# B&R Automation Studio project PrintMarkLabWork
Automation Studio 4.12.4.107 SP; technology packages: Acp10Arnc0 5.23.1, mapp 5.23.1, mappView 5.23.0

## Configuration Config1

CPU X20CP0484, AutomationRuntime G4.93, Build 4.1.2, Vc V4.73.0

### Task classes (Cpu.sw)
```
Cyclic#1 (cycle 2000 us, tolerance 10000 us):
  AutoCtrl <- Source.AutoCtrl.AutoCtrl.prg  // Auto Ctrl Logic
  ConvCtrl <- Source.AxisConf.ConvCtrl.prg  // Conv Ctrl Logic
  CutterCtrl <- Source.AxisConf.CutterCtrl.prg  // Cutter Ctrl Logic
Cyclic#4 (cycle 100000 us, tolerance 100000 us):
  Alarm <- InfraStructure.Alarm.Alarm.prg  // Alarm Logic
Cyclic#7 (cycle 1000000 us, tolerance 1000000 us):
  Visu <- InfraStructure.Visu.Visu.prg  // Visu Logic
DataObjects: Acp10sys
NcDataObjects: acp10etxen <- Axis.acp10etxen.dob, gAxis01a <- Axis.gAxis01obj.gAxis01a.dob, gAxis01i <- Axis.gAxis01obj.gAxis01i.dob, gAxis02a <- Axis.gAxis02obj.gAxis02a.dob, gAxis02i <- Axis.gAxis02obj.gAxis02i.dob
Binaries: arsvcreg, udbdef, mvLoader, FWRules, TCData, TCLang, arflatprv, arcoal, Acp10map, acp10cfg, SlaveAxis, ashwac, User, sysconf, asfw, arconfig, ashwd, MasterAxis, iomap, Role, DataRConf, AlarmConf, UserConf, User_1, TC
Libraries: Acp10man, Acp10par, NcGlobal, Acp10_MC, sys_lib, brsystem, runtime, MpAxis, MpBase, MpCom, MpServer, MC_RegMa, MpAlarmX, astime, MpData, FileIO, DataObj, MpUserX, arssl, asieccon, powerlnk, asbrstr, aruser, arcert, aseth, ashw
```

### Hardware
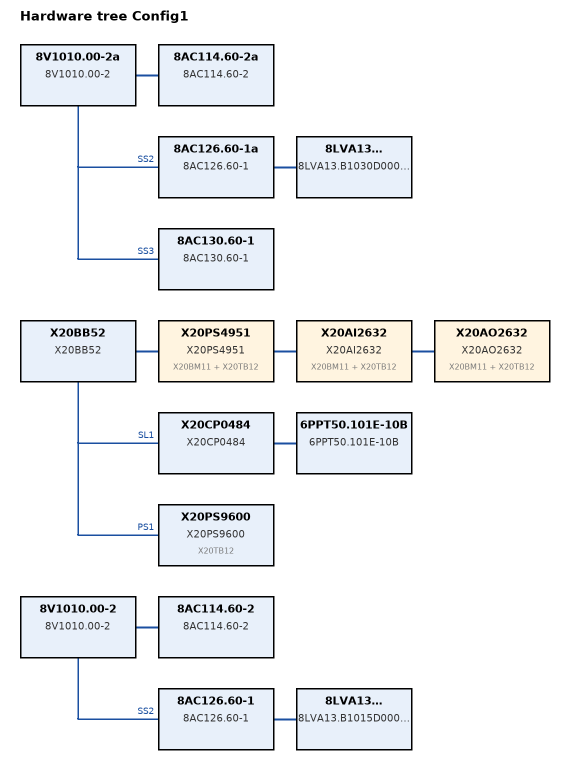
```
6PPT50.101E-10B : 6PPT50.101E-10B v1.3.8.0  [ETH1 -> X20CP0484.IF2 [Cable Type=PowerlinkCable, Length=10, Version=1.0.0.3]]
  Terminal = true
  Startmode = 2
  ShowBootlogoWeb = 1
  TimeZone = 250
  PasswordVNC = 
  BrowserVKeyboard = 0
  PasswordCIFS = 
  PasswordService = 
8AC114.60-2 : 8AC114.60-2 v1.0.0.8  [SS -> 8V1010.00-2.SS1; PLK1 -> X20CP0484.IF3 (NodeNumber=1) [Cable Type=PowerlinkCable, Length=10, Version=1.0.0.3]; PLK2 -> 8AC114.60-2a.PLK1 (NodeNumber=1) [Cable Type=PowerlinkCable, Length=10, Version=1.0.0.3]]
8AC114.60-2a : 8AC114.60-2 v1.0.0.8  [SS -> 8V1010.00-2a.SS1; PLK1 -> 8AC114.60-2.PLK2 (NodeNumber=2) [Cable Type=PowerlinkCable, Length=10, Version=1.0.0.3]]
8AC126.60-1 : 8AC126.60-1 v2.2.0.0  [SS -> 8V1010.00-2.SS2]
8AC126.60-1a : 8AC126.60-1 v2.2.0.0  [SS -> 8V1010.00-2a.SS2]
8AC130.60-1 : 8AC130.60-1 v2.2.0.0  [SS -> 8V1010.00-2a.SS3]
8LVA13.B1015D000-0 : 8LVA13.B1015D000-0 v2.2.0.3  [EC -> 8AC126.60-1.EC; MT -> 8V1010.00-2.MT1]
8LVA13.B1030D000-0 : 8LVA13.B1030D000-0 v2.2.0.3  [EC -> 8AC126.60-1a.EC; MT -> 8V1010.00-2a.MT1]
8V1010.00-2 : 8V1010.00-2 v2.2.0.0
  MotionTP = Acp10Arnc0
  SinglePhaseOperation = on
  BothEndSwitchesAreNormallyOpen_r1 = on
  QuickStopIsNormallyOpen_r1 = on
8V1010.00-2a : 8V1010.00-2 v2.2.0.0
  MotionTP = Acp10Arnc0
  SinglePhaseOperation = on
  AxisIsPeriodic_r1 = on
  Period_r1 = 3600
  BothEndSwitchesAreNormallyOpen_r1 = on
  QuickStopIsNormallyOpen_r1 = on
X20AI2632 : X20AI2632 v1.3.0.0  [SS1 -> X20TB12b.SS; SL -> X20BM11a.SL1]
  Supervision = off
X20AO2632 : X20AO2632 v1.2.0.0  [SS1 -> X20TB12c.SS; SL -> X20BM11b.SL1]
  Supervision = off
X20BB52 : X20BB52 v1.2.0.0
X20BM11 : X20BM11 v1.1.0.0  [X2X1 -> X20BB52.IF6]
X20BM11a : X20BM11 v1.1.0.0  [X2X1 -> X20BM11.X2X2]
X20BM11b : X20BM11 v1.1.0.0  [X2X1 -> X20BM11a.X2X2]
X20CP0484 : X20CP0484 v1.6.0.0  [SL -> X20BB52.SL1]
  Connector IF2:
    ActivateDevice = 1
    Mode = Manual
    InternetAddress = 10.91.10.142
    SubnetMask = 255.255.255.0
    ActivateSnmp = 2
  ConfigurationID = PrintMarkLabWork_Config1
  Simulation = 1
  TimerDeviceType = EPLX2X
  TimerDevice = X20CP0484.IF3
  TaskClassIdleTime = 2000
  Cyclic1Duration = 2000
  Cyclic1Tolerance = 10000
  Cyclic2Duration = 20000
  Cyclic2Tolerance = 20000
  Cyclic3Duration = 50000
  Cyclic3Tolerance = 50000
  Cyclic4Duration = 100000
  Cyclic4Tolerance = 100000
  Cyclic5Duration = 200000
  Cyclic5Tolerance = 200000
  Cyclic6Duration = 500000
  Cyclic6Tolerance = 500000
  Cyclic7Duration = 1000000
  Cyclic7Tolerance = 1000000
  Cyclic8Duration = 10000
  Cyclic8Tolerance = 30000000
  FileDevice1
  FileDeviceName1 = USER
  FileDevicePath1 = USER_PATH
  ActivateOpcUa = 1
  OpcUaInformationModels_PV_Version = 1
X20PS4951 : X20PS4951 v1.2.0.0  [SS1 -> X20TB12a.SS; SL -> X20BM11.SL1]
  Supervision = off
X20PS9600 : X20PS9600 v1.6.0.0  [PS -> X20BB52.PS1; SS1 -> X20TB12.SS]
X20TB12 : X20TB12 v1.0.0.0
X20TB12a : X20TB12 v1.0.0.0
X20TB12b : X20TB12 v1.0.0.0
X20TB12c : X20TB12 v1.0.0.0
```

### Acp10cfg.ncc - X20CP0484/Motion/Acp10cfg.ncc
```
NcConfiguration (Version=5.23.1, NcSwId=Acp10)
  ACP10CF1_typ:
    cnt_nettrc_rec_drive = 1500
    bufsize_trace_upload = 1200
    tc_nc_man_task = Cyclic #1
    glob_pv_as_ncobject = Yes
    ncsys_dl_broadcast = Yes
    ncsys_dl_acp_reset = Yes
    safemc_log_err_to_ax = Yes
    network_init:
      ncsw_init_execute = Yes
      automatic_execute = No
      node_nr_warning = Yes
      net_err_before_ncact = Yes
    nettrc:
      enter_parsecrec = Yes
      enter_ncaction = Yes
      save_ring_startidx = Yes
    cam_prof_download:
      cam_dat_dl_parallel = No
      tc_cam_dl_parallel = Task class for NC Manager task
    plk_if[0]:
      if_name = IF3
      tc_CycDat_PLCopen = Task class for NC Manager task
      mc_broadcast_extdat = No
```

### Acp10map.ncm - X20CP0484/Motion/Acp10map.ncm
```
NcMapping (NcSwId=Acp10, DisabledNodesAreHidden=False)
  NcObject gAxis01 (ModuleId=8V1010.00-2, Type=ncAXIS, Channel=1, AcoposSimulation=Off, InitParameter=gAxis01i, AcoposParameter=gAxis01a, Disabled=FALSE, ModuleDisabled=FALSE)
  NcObject 8V1010.00-2_ncV_AXIS1 (ModuleId=8V1010.00-2, Type=ncV_AXIS, Channel=1, Disabled=TRUE, ModuleDisabled=FALSE)
  NcObject gAxis02 (ModuleId=8V1010.00-2a, Type=ncAXIS, Channel=1, AcoposSimulation=Off, InitParameter=gAxis02i, AcoposParameter=gAxis02a, AdditionalData=PLCopen_ModPos="3600,1" , Disabled=FALSE, ModuleDisabled=FALSE)
  NcObject 8V1010.00-2a_ncV_AXIS1 (ModuleId=8V1010.00-2a, Type=ncV_AXIS, Channel=1, Disabled=TRUE, ModuleDisabled=FALSE)
```

### MasterAxis.mpaxisbasic - X20CP0484/Motion/MasterAxis.mpaxisbasic
```
Element gAxisMaster (Type=mpaxisbasic)
  Alarms = MpAlarmX
```

### SlaveAxis.mpaxisbasic - X20CP0484/Motion/SlaveAxis.mpaxisbasic
```
Element gAxisSlave (Type=mpaxisbasic)
  Alarms = MpAlarmX
```

### AlarmConf.mpalarmxcore - X20CP0484/mappServices/Alarm/AlarmConf.mpalarmxcore
```
Element gAlarmXMain (Type=mpalarmxcore)
  mapp.AlarmX.Core.Configuration:
    [0]:
      Name = InCuttingZone
      Message = Cutter is in Cutting Zone. Please Remove the Cutter
      Code = 50
      Severity = 10
      Behavior = PersistentAlarm
        ReactionUntilAcknowledged = FALSE
    [1]:
      Name = CuttingError
      Message = Product without Print Mark Exceeded Limit
      Code = 80
      Severity = 50
      Behavior = PersistentAlarm
        ReactionUntilAcknowledged = FALSE
```

### DataRConf.mpdatarecorder - X20CP0484/mappServices/DataRecorder/DataRConf.mpdatarecorder
```
Element gDataRecorder (Type=mpdatarecorder)
  Alarms = MpAlarmX
```

### UserConf.mpuserx - X20CP0484/mappServices/User/UserConf.mpuserx
```
Element UserMgmtX (Type=mpuserx)
  ServerSettings:
    Server:
      AdditionalUserData:
        [0] = mail
        [1] = telephoneNumber
  Users:
    DefUser#1:
      id = Admin
      name = Administrator
      lang = en
    DefUser#2:
      id = Operator
      name = Machine Operator
      lang = en
    DefUser#3:
      id = Anonymous
  Groups:
    DefGroup#1:
      id = Administrators
      level = 100
      admin = TRUE
      rights:
        [0] = FullAccess
    DefGroup#2:
      id = Operator
      level = 50
```

## Logical view

Binary libraries used (declarations not repeated): operator, runtime, astime, AsIecCon, Acp10man 5.23.1, Acp10par 5.23.1, NcGlobal 5.23.1, Acp10_MC 5.23.1, sys_lib, brsystem, MpAxis 1.86.0, MpBase, MpCom 5.23.1, MpServer, MC_RegMa 5.23.1, MpAlarmX 5.23.1, MpData 5.23.1, FileIO, DataObj, MpUserX 5.23.1

### Global.var - Global variables
```iecst
(*********************************************************************************
 * Copyright: B&R Industrial Automation GmbH
 * Author:    kasliwals
 * Created:   December 17, 2023/12:04 AM
 *********************************************************************************)
(*Axis Variables*)
VAR
	gAxis01 : ACP10AXIS_typ; (*Master Axis*)
	gAxis02 : ACP10AXIS_typ; (*Slave Axis*)
END_VAR
(*Axis Global structure*)
VAR
	gAx_Slave : AxisBasic_type; (*Slave Axis Structure*)
	gAx_Master : AxisBasic_type; (*MAster axis Structure*)
END_VAR
(*HMI Variables*)
VAR
	gMI_ModeConfirm : BOOL; (*Mode Confirm VA*)
	gMI_MODE : BOOL; (*Mode VA*)
END_VAR
```


### Package Logical/Axis - Axis Package

### Package Logical/Axis/gAxis01obj - gAxis01obj

### gAxis01i.ax
```
InitParameter (Version=5.23.1, NcSwId=ACP10)
  ACP10AXIS_typ:
    dig_in:
      level:
        reference = ncACTIV_HI
        pos_hw_end = ncACTIV_HI
        neg_hw_end = ncACTIV_HI
        trigger1 = ncACTIV_HI
        trigger2 = ncACTIV_HI
    encoder_if:
      parameter:
        count_dir = ncSTANDARD
        scaling:
          load:
            units = 1600
            rev_motor = 1
    limit:
      parameter:
        v_pos = 10000.0
        v_neg = 10000.0
        a1_pos = 50000.0
        a2_pos = 50000.0
        a1_neg = 50000.0
        a2_neg = 50000.0
        t_jolt = 0.0
        t_in_pos = 0.0
        pos_sw_end = 8388607
        neg_sw_end = -8388608
        ds_warning = 500.0
        ds_stop = 1000.0
        a_stop = 1.0E+30
        dv_stop = 0.0
        dv_stop_mode = ncOFF
    controller:
      mode = ncPOSITION + ncFF
      position:
        kv = 262.0
        tn = 0.0
        t_predict = 0.0004
        t_total = 0.0004
        p_max = 1.0E+30
        i_max = 0.0
      speed:
        kv = 0.55
        tn = 0.0
        t_filter = 0.0
        isq_filter1:
          type = ncOFF
          a0 = 0.0
          a1 = 0.0
          b0 = 0.0
          b1 = 0.0
          b2 = 0.0
          c0_par_id = 0
          c1_par_id = 0
        isq_filter2:
          type = ncOFF
          a0 = 0.0
          a1 = 0.0
          b0 = 0.0
          b1 = 0.0
          b2 = 0.0
          c0_par_id = 0
          c1_par_id = 0
        isq_filter3:
          type = ncOFF
          a0 = 0.0
          a1 = 0.0
          b0 = 0.0
          b1 = 0.0
          b2 = 0.0
          c0_par_id = 0
          c1_par_id = 0
      uf:
        type = ncLINEAR + ncCORRECTION
        auto_config = ncMOTOR_PAR
        u0 = 0.0
        un = 0.0
        fn = 50.0
        k_f_slip = 0.0
      ff:
        mode = ncSTANDARD
        torque_load = 0.0
        torque_pos = 0.0
        torque_neg = 0.0
        kv_torque = 0.0117175
        inertia = 8.74906E-05
        t_filter_a = 0.0
      fb:
        mode = ncSTANDARD
        speed_mix_ratio = 0.0
        speed_kv = 0.0
      model:
        mass1:
          inertia = 0.0
          viscous_friction = 0.0
        mass2:
          inertia = 0.0
          viscous_friction = 0.0
          stiffness = 0.0
          damping = 0.0
    move:
      stop:
        parameter[0]:
          decel_ramp = ncA_LIMIT
          controller = ncON
        parameter[1]:
          decel_ramp = ncA_LIMIT
          controller = ncON
        parameter[2]:
          decel_ramp = ncA_LIMIT
          controller = ncON
        parameter[3]:
          decel_ramp = ncA_LIMIT
          controller = ncON
        quickstop:
          decel_ramp = ncA_LIMIT
          t_jolt = 0.0
        drive_error:
          decel_ramp = ncA_LIMIT
      homing:
        parameter:
          s = 0
          v_switch = 5000.0
          v_trigger = 500.0
          a = 50000.0
          mode = ncDIRECT
          edge_sw = ncPOSITIVE
          start_dir = ncPOSITIVE
          trigg_dir = ncPOSITIVE
          ref_pulse = ncOFF
          fix_dir = ncOFF
          tr_s_block = 0.0
          torque_lim = 0.0
          ds_block = 0.0
          ds_stop = 0.0
      basis:
        parameter:
          v_pos = 500.0
          v_neg = 5000.0
          a1_pos = 50000.0
          a2_pos = 50000.0
          a1_neg = 50000.0
          a2_neg = 50000.0
    message:
      text:
        parameter:
          format = ncBREAK + ncZERO
          columns = 80
          data_modul = acp10etxen
```

### Package Logical/Axis/gAxis02obj - gAxis02obj

### gAxis02i.ax
```
InitParameter (Version=5.23.1, NcSwId=ACP10)
  ACP10AXIS_typ:
    dig_in:
      level:
        reference = ncACTIV_HI
        pos_hw_end = ncACTIV_HI
        neg_hw_end = ncACTIV_HI
        trigger1 = ncACTIV_HI
        trigger2 = ncACTIV_HI
    encoder_if:
      parameter:
        count_dir = ncSTANDARD
        scaling:
          load:
            units = 3600
            rev_motor = 1
    limit:
      parameter:
        v_pos = 108000.0
        v_neg = 108000.0
        a1_pos = 1080000.0
        a2_pos = 1080000.0
        a1_neg = 1080000.0
        a2_neg = 1080000.0
        t_jolt = 0.18
        t_in_pos = 0.0
        pos_sw_end = 8388607
        neg_sw_end = -8388608
        ds_warning = 180.0
        ds_stop = 360.0
        a_stop = 1.0E+30
        dv_stop = 0.0
        dv_stop_mode = ncOFF
    controller:
      mode = ncPOSITION + ncFF
      position:
        kv = 241.0
        tn = 0.0
        t_predict = 0.0004
        t_total = 0.0004
        p_max = 1.0E+30
        i_max = 0.0
      speed:
        kv = 0.55
        tn = 0.0
        t_filter = 0.0
        isq_filter1:
          type = ncOFF
          a0 = 0.0
          a1 = 0.0
          b0 = 0.0
          b1 = 0.0
          b2 = 0.0
          c0_par_id = 0
          c1_par_id = 0
        isq_filter2:
          type = ncOFF
          a0 = 0.0
          a1 = 0.0
          b0 = 0.0
          b1 = 0.0
          b2 = 0.0
          c0_par_id = 0
          c1_par_id = 0
        isq_filter3:
          type = ncOFF
          a0 = 0.0
          a1 = 0.0
          b0 = 0.0
          b1 = 0.0
          b2 = 0.0
          c0_par_id = 0
          c1_par_id = 0
      uf:
        type = ncLINEAR + ncCORRECTION
        auto_config = ncMOTOR_PAR
        u0 = 0.0
        un = 0.0
        fn = 50.0
        k_f_slip = 0.0
      ff:
        mode = ncSTANDARD
        torque_load = 0.0
        torque_pos = 0.0
        torque_neg = 0.0
        kv_torque = 0.00398844
        inertia = 0.00010255
        t_filter_a = 0.0
      fb:
        mode = ncSTANDARD
        speed_mix_ratio = 0.0
        speed_kv = 0.0
      model:
        mass1:
          inertia = 0.0
          viscous_friction = 0.0
        mass2:
          inertia = 0.0
          viscous_friction = 0.0
          stiffness = 0.0
          damping = 0.0
    move:
      stop:
        parameter[0]:
          decel_ramp = ncA_LIMIT
          controller = ncON
        parameter[1]:
          decel_ramp = ncA_LIMIT
          controller = ncON
        parameter[2]:
          decel_ramp = ncA_LIMIT
          controller = ncON
        parameter[3]:
          decel_ramp = ncA_LIMIT
          controller = ncON
        quickstop:
          decel_ramp = ncA_LIMIT
          t_jolt = 0.0
        drive_error:
          decel_ramp = ncA_LIMIT
      homing:
        parameter:
          s = 0
          v_switch = 5000.0
          v_trigger = 500.0
          a = 50000.0
          mode = ncDIRECT
          edge_sw = ncPOSITIVE
          start_dir = ncPOSITIVE
          trigg_dir = ncPOSITIVE
          ref_pulse = ncOFF
          fix_dir = ncOFF
          tr_s_block = 0.0
          torque_lim = 0.0
          ds_block = 0.0
          ds_stop = 0.0
      basis:
        parameter:
          v_pos = 500.0
          v_neg = 5000.0
          a1_pos = 50000.0
          a2_pos = 50000.0
          a1_neg = 50000.0
          a2_neg = 50000.0
    message:
      text:
        parameter:
          format = ncBREAK + ncZERO
          columns = 80
          data_modul = acp10etxen
```

### Package Logical/Source - Source Package

### Package Logical/Source/AutoCtrl - Auto Ctrl Package

### Program Logical/Source/AutoCtrl/AutoCtrl (IEC) - Auto Ctrl task

#### Main.st - Init, cyclic, exit code
```iecst
(*********************************************************************************
 * Copyright: B&R Industrial Automation GmbH
 * Author:    kasliwals
 * Created:   December 16, 2023/11:35 PM
* Description: Auto Ctrl Logic for Print Marl
* Version : 1.0.0.0
 *********************************************************************************)

PROGRAM _INIT
	(* Insert code here *)
	Status_CutterCtrl := PV_xgetadr(ADR('CutterCtrl:iCutterCtrl'),ADR(CutterAdd),ADR(SizeCutter));
	Status_ConvCtrl := PV_xgetadr(ADR('ConvCtrl:iConvCtrl'),ADR(ConvAdd),ADR(SizeConv));
	Status_CamSeq := PV_xgetadr(ADR('CutterCtrl:iAx_CamSeq'),ADR(CamAdd),ADR(SizeCam));
	Status_RegCapture := PV_xgetadr(ADR('CutterCtrl:iFb_RegCapture'),ADR(RegAdd),ADR(RegSize));
	gAx_Master.In.Enable := TRUE;
	gAx_Slave.In.Enable := TRUE;
	iMI_CurrentMode := 'Manual Mode';
END_PROGRAM

PROGRAM _CYCLIC
	(* Insert code here *)
	pCutterCtrl ACCESS CutterAdd;
	pConvCtrl ACCESS ConvAdd;
 	pAx_CamSeq ACCESS CamAdd;
	pRegCapture ACCESS RegAdd;

	CASE AutoCtrlState OF
		WAIT :
			iMI_MachineStatus := 'Please Select the Mode And Then Press Start';
			gAx_Master.In.Enable := TRUE;
			gAx_Slave.In.Enable := TRUE;

			IF iAutoCtrl.Cmd.Start THEN
				pConvCtrl.Cmd.Start := TRUE;
				pCutterCtrl.Cmd.Start := TRUE;
				AutoCtrlState := MODE_SELECT;
			END_IF

		MODE_SELECT :
			IF gMI_ModeConfirm THEN

				IF iAutoCtrl.Cmd.AutoMode THEN
					iMI_CurrentMode := 'Auto Mode';
					AutoCtrlState := HOMING_DONE;
				ELSE
					iMI_CurrentMode := 'Manual Mode';
					AutoCtrlState := MANUAL_START;
				END_IF
			END_IF
		HOMING_DONE :
			iMI_MachineStatus := 'Homing Both Axis';
			pAx_CamSeq.In.ErrorReset := TRUE;

			IF gAx_Master.Out.IsHomed AND gAx_Slave.Out.IsHomed THEN
				pAx_CamSeq.In.ErrorReset := FALSE;
				AutoCtrlState := AUTO_START;
			END_IF

		AUTO_START :

			IF pAx_CamSeq.Out.Info.MasterReady AND pAx_CamSeq.Out.Info.SlaveReady AND pAx_CamSeq.Out.StatusID = 0 THEN

				pAx_CamSeq.In.StartSequence := TRUE;
			END_IF
			IF pAx_CamSeq.Out.StatusID <> 0 THEN
				pAx_CamSeq.In.ErrorReset := TRUE;
				pAx_CamSeq.In.ErrorReset := FALSE;
			END_IF

			IF pAx_CamSeq.Out.InSync AND iAutoCtrl.Cmd.Start THEN
				iMI_MachineStatus := 'Running in Auto Mode';
				gAx_Master.In.MoveVelocity := TRUE;
			END_IF

			IF iAutoCtrl.Cmd.Stop THEN
				iMI_MachineStatus := 'Stop Pressed. Press Start to Restart Or Change mode to Exit Mode and select mode.';
				gAx_Master.In.MoveVelocity := FALSE;
			END_IF

			IF iAutoCtrl.Cmd.DisableCutter THEN
				iMI_MachineStatus := 'Cutter Disabled Pressed';
				pAx_CamSeq.In.StartSequence := FALSE;
				pCutterCtrl.Cmd.Start := FALSE;
				gAx_Slave.In.Power := FALSE;
				AutoCtrlState := CUTTER_DISABLED_HOME;
			END_IF

			IF iAutoCtrl.Cmd.ChangeMode AND iAutoCtrl.Cmd.Stop THEN
				iMI_MachineStatus := 'Machine Stopped';
				gAx_Master.In.MoveVelocity := FALSE;
				iAutoCtrl.Cmd.ChangeMode := FALSE;
				pAx_CamSeq.In.StartSequence := FALSE;
				AutoCtrlState := STOP;
			END_IF
		CUTTER_DISABLED_HOME :
				iMI_MachineStatus := 'Homing Cutter';
			gAx_Slave.In.Power := TRUE;
			pCutterCtrl.Cmd.Start := TRUE;
			AutoCtrlState := CUTTER_DISABLED;
		CUTTER_DISABLED :
			IF gAx_Slave.Out.IsHomed THEN
				iMI_MachineStatus := 'Cutter Disbaled. Stop Mode or Restart Cutter Again';
				gAx_Slave.In.Home := FALSE;
			END_IF
			IF iAutoCtrl.Cmd.Stop THEN
				gAx_Master.In.MoveVelocity := FALSE;
			END_IF
			IF iAutoCtrl.Cmd.Start THEN
				gAx_Master.In.MoveVelocity := TRUE;
			END_IF
			IF iAutoCtrl.Cmd.DisableCutter = FALSE THEN
				iMI_MachineStatus := 'Cutter Enabled';
				AutoCtrlState := AUTO_START;
			END_IF
			IF iAutoCtrl.Cmd.ChangeMode AND iAutoCtrl.Cmd.Stop THEN
				iMI_MachineStatus := 'Machine Stopped';
				gAx_Master.In.MoveVelocity := FALSE;
				iAutoCtrl.Cmd.ChangeMode := FALSE;
				pAx_CamSeq.In.StartSequence := FALSE;
				AutoCtrlState := STOP;
			END_IF

		MANUAL_START :
			IF iAutoCtrl.Cmd.Stop AND iAutoCtrl.Cmd.ChangeMode THEN
				iMI_MachineStatus := 'Machine Stopped';
				iAutoCtrl.ManualCmd.ConvPowerON := FALSE;
				iAutoCtrl.ManualCmd.CutterPowerON := FALSE;
				AutoCtrlState := STOP;
			END_IF

		STOP :
			iMI_MachineStatus := 'Machine Stopped';
			iAutoCtrl.Cmd.Start := FALSE;
			gMI_ModeConfirm := FALSE;
			gAx_Master.In.Power := FALSE;
			gAx_Slave.In.Power := FALSE;
			gAx_Master.In.Enable := FALSE;
			gAx_Slave.In.Enable := FALSE;
			pConvCtrl.Cmd.Start := FALSE;
			iAutoCtrl.Cmd.ChangeMode := FALSE;
			pCutterCtrl.Cmd.Start := FALSE;
			iAutoCtrl.Cmd.DisableCutter := FALSE;
			iAutoCtrl.Cmd.Stop := FALSE;
			AutoCtrlState := WAIT;

		IN_CUTTING_ZONE :
			iMI_MachineStatus := 'Cutter In Cutting Zone.';
			iAutoCtrl.ManualCmd.ConvPowerON := FALSE;
			iAutoCtrl.ManualCmd.CutterPowerON := FALSE;
			iAutoCtrl.ManualCmd.ConvHome := FALSE;
			iAutoCtrl.ManualCmd.CutterHome := FALSE;
			IF gAx_Slave.Out.Position > UPPER_CUT_POS OR gAx_Slave.Out.Position <LOWER_CUT_POS  THEN
				iAutoCtrl.Cmd.Start := FALSE;
				AutoCtrlState := WAIT;
			END_IF
		END_CASE

	IF NOT iAutoCtrl.Cmd.AutoMode THEN
		gAx_Master.In.Power := iAutoCtrl.ManualCmd.ConvPowerON;
		gAx_Slave.In.Power := iAutoCtrl.ManualCmd.CutterPowerON;
		gAx_Master.In.JogNegative := pConvCtrl.Cmd.JogBack;
		gAx_Master.In.JogPositive := pConvCtrl.Cmd.JogFwd;
		gAx_Slave.In.JogNegative := pCutterCtrl.Cmd.JogBack;
		gAx_Slave.In.JogPositive := pCutterCtrl.Cmd.JogFwd;

	END_IF

	pConvCtrl.Cmd.AutoMode := iAutoCtrl.Cmd.AutoMode;
	pCutterCtrl.Cmd.AutoMode := iAutoCtrl.Cmd.AutoMode;
	IF gAx_Slave.Out.Position < UPPER_CUT_POS AND gAx_Slave.Out.Position > LOWER_CUT_POS AND NOT iAutoCtrl.Cmd.AutoMode THEN
		AutoCtrlState := IN_CUTTING_ZONE;
	END_IF

	iMI_LastBagLen := pRegCapture.AdditionalInfo.ActLength / TEN;
	iMI_AvgBagLen := pRegCapture.AdditionalInfo.AverageProductLength /TEN;
	IF iAutoCtrl.Cmd.AutoMode THEN
		iMI_CurrentMode := 'Auto Mode';

	ELSE
		iMI_CurrentMode := 'Manual Mode';
	END_IF

	gMI_MODE := iAutoCtrl.Cmd.AutoMode;

END_PROGRAM

PROGRAM _EXIT
	(* Insert code here *)

END_PROGRAM
```

#### Types.typ - Local data types
```iecst
(*********************************************************************************
 * Copyright: B&R Industrial Automation GmbH
 * Author:    kasliwals
 * Created:   December 16, 2023/11:35 PM
 *********************************************************************************)

TYPE
	AutoCtrl_enum :
		( (*Auto Ctrl State*)
		WAIT, (*Wait state*)
		MODE_SELECT, (*Mode Select state*)
		HOMING_DONE, (*homing State*)
		MANUAL_START, (*Manual Mode*)
		AUTO_START, (*Auto mode state*)
		STOP, (*Stop state*)
		MANUAL_JOGF, (*Manual jog f State*)
		MANUAL_JOGN, (*Manual jog N State*)
		IN_CUTTING_ZONE, (*Cutting zone state*)
		CUTTER_DISABLED, (*Cutter Disabled STate*)
		CUTTER_DISABLED_HOME (*Cutter Homing after disable*)
		);
END_TYPE
```

#### Variables.var - Local variables
```iecst
(*********************************************************************************
 * Copyright: B&R Industrial Automation GmbH
 * Author:    kasliwals
 * Created:   December 16, 2023/11:35 PM
 *********************************************************************************)
(*Status and address Variables for Pointers*)
VAR
	Status_CutterCtrl : UINT; (*Status*)
	CutterAdd : UDINT; (*Address*)
	SizeCutter : UDINT; (*Size*)
	Status_CamSeq : UINT; (*Status*)
	SizeCam : UDINT; (*Size*)
	CamAdd : UDINT; (*Address*)
	Status_ConvCtrl : UINT; (*Statsus*)
	RegAdd : UDINT; (*Address*)
	Status_RegCapture : UINT; (*Status*)
	RegSize : UDINT; (*Size*)
	ConvAdd : UDINT; (*Address*)
	SizeConv : UDINT; (*Address*)
END_VAR
(*Pointer Variables*)
VAR
	pCutterCtrl : REFERENCE TO AxisCtrl_typ; (*Pointer to conv ctrl*)
	pRegCapture : REFERENCE TO MC_BR_RegMarkCapture002; (*Pointer to reg capture*)
	pConvCtrl : REFERENCE TO AxisCtrl_typ; (*Pointer to Conv Ctrl*)
	pAx_CamSeq : REFERENCE TO AxisCamSeqMain_Typ; (*Pointer cam seq*)
END_VAR
(*Process Variables*)
VAR
	AutoCtrlState : AutoCtrl_enum; (*Auto control state*)
	iAutoCtrl : AutoCtrl_typ; (*Auto ctrl struture*)
END_VAR
(*Constants*)
VAR CONSTANT
	UPPER_CUT_POS : LREAL := 3013; (*Upper cut limit*)
	PROUCT_WITHOUT_RM : INT := 5; (*Limit of products without PM*)
	TEN : REAL := 10; (*TEN number*)
	LOWER_CUT_POS : LREAL := 2653; (*Lower Cutting Limit*)
END_VAR
(*HMI Variables*)
VAR
	iMI_LastBagLen : REAL; (*Last bag length*)
	iMI_AvgBagLen : REAL; (*Avg Bag length*)
	iMI_CurrentMode : STRING[80]; (*Current Mode*)
	iMI_MachineStatus : STRING[100];
END_VAR
```

#### Alarm.st - Alarm action
```iecst
(*********************************************************************************
 * Copyright: B&R Industrial Automation GmbH
 * Author:    kasliwals
 * Created:   December 16, 2023/11:54 PM
* Description: Alarm Logic
* Version : 1.0.0.0
 *********************************************************************************)

ACTION Alarm:
	IF gAx_Slave.Out.Position < UPPER_CUT_POS AND gAx_Slave.Out.Position > LOWER_CUT_POS THEN
		MpAlarmXSet(gAlarmXMain,'InCuttingZone');
	ELSE
		MpAlarmXReset(gAlarmXMain,'InCuttingZone');
	END_IF

	IF pRegCapture.ProductsWithoutRM > PROUCT_WITHOUT_RM THEN
		MpAlarmXSet(gAlarmXMain,'CuttingError');
		AutoCtrlState := STOP;
	ELSE
		MpAlarmXReset(gAlarmXMain,'CuttingError');
	END_IF

END_ACTION
```

### AutoCtrlTyp.typ - Auto ctrl global types
```iecst
(*********************************************************************************
 * Copyright: B&R Industrial Automation GmbH
 * Author:    kasliwals
 * Created:   December 16, 2023/11:35 PM
 *********************************************************************************)

TYPE
	AutoCmd_typ : 	STRUCT  (*Auto Ctrl Command Type*)
		Start : BOOL; (*Start cmd*)
		Stop : BOOL; (*Stop cmd*)
		AutoMode : BOOL; (*Auto Mode cmd*)
		ChangeMode : BOOL; (*Change Mode cmd*)
		DisableCutter : BOOL; (*Disable Cutter cmd*)
	END_STRUCT;
	AutoPara_typ : 	STRUCT  (*Auto Ctrl Para Type*)
		ConvSpeed : REAL; (*Conv speed Para*)
		ConvJogSpeed : REAL; (*Conv Jog SPeed*)
		CutterJogSpeed : REAL; (*Cutter Jog Speed*)
	END_STRUCT;
	AutoManCmd_typ : 	STRUCT  (*Auto Ctrl Manaual Cmd Type*)
		ConvPowerON : BOOL; (*Conv power on*)
		CutterPowerON : BOOL; (*Cutter Power On*)
		CutterHome : BOOL; (*Cutter Home cmd*)
		ConvHome : BOOL; (*Conv home cmd*)
	END_STRUCT;
	AutoCtrl_typ : 	STRUCT  (*Auto Ctrl Type*)
		Cmd : AutoCmd_typ; (*Auto Ctrl cmd type*)
		Para : AutoPara_typ; (*Auto Ctrl Para type*)
		ManualCmd : AutoManCmd_typ; (*Auto Ctrl Manual Cmd Type*)
	END_STRUCT;
END_TYPE
```

### Package Logical/Source/AxisConf - Axis Config Package

### Program Logical/Source/AxisConf/CutterCtrl (IEC) - Cutter Ctrl Task

#### Main.st - Init, cyclic, exit code
```iecst
(*********************************************************************************
 * Copyright: B&R Industrial Automation GmbH
 * Author:    kasliwals
 * Created:   December 11, 2023/10:45 AM
* Description: Cam Sequencer Logic for Master and Slave Movement
* Version : 1.0.0.0
 *********************************************************************************)

PROGRAM _INIT
	gAx_Slave.In.Parameters.Jog.Acceleration := 108000;
	gAx_Slave.In.Parameters.Jog.Deceleration := 1080000;
	gAx_Slave.In.Parameters.Jog.Velocity := 360;

	iVa_RegCaptureAdvPara.EventSourceParID := ACP10PAR_STAT_TRIGGER1;
	iVa_RegCaptureAdvPara.Edge := ncP_EDGE;
	iVa_RegCaptureAdvPara.MinWidth := 50;
	iVa_RegCaptureAdvPara.MaxWidth := 200;
	iVa_RegCaptureAdvPara.WindowNeg := 200;
	iVa_RegCaptureAdvPara.WindowPos := 200;
	iVa_RegCaptureAdvPara.SensorDelay := 200;
	iVa_RegCaptureAdvPara.CorrectCurrentCycle := TRUE;
	iVa_RegCaptureAdvPara.CorrectionValueLimitNeg := 70;
	iVa_RegCaptureAdvPara.CorrectionValueLimitPos := 70;

	iVa_RegCaptureConfig.DistanceToSensor := 1050;
	iVa_RegCaptureConfig.ProductLength := 700;
	iVa_RegCaptureConfig.RegMarkPosition := 700;
	iVa_RegCaptureConfig.RegMarkOffset := 10;

END_PROGRAM

PROGRAM _CYCLIC

	SingleCam;
	RegCapture;
	SingleCutter;
	Mapping;
END_PROGRAM

PROGRAM _EXIT
	(* Insert code here *)
	iFb_MpAxisBasic.Enable := FALSE;
	iFb_MpAxisBasic();
	iFb_MpAxisSlave.Enable := FALSE;
	iFb_MpAxisSlave();
	iFb_CamSeq.Enable := FALSE;
	iFb_CamSeq();
END_PROGRAM
```

#### Types.typ - Local data types
```iecst
(*********************************************************************************
 * Copyright: B&R Industrial Automation GmbH
 * Author:    kasliwals
 * Created:   December 16, 2023/11:36 PM
 *********************************************************************************)

TYPE
	AxisState_enum :
		( (*Axis States*)
		WAIT, (*Wait State*)
		ACTIVE, (*Active State*)
		POWER_ON, (*Power on state*)
		POSITIVE_HOMING_MODE, (*Positive side homing*)
		NEGATIVE_HOMING_MODE, (*Negative side homing*)
		HOMING, (*Homing*)
		AUTO_MODE, (*Auto mode state*)
		OPERATION, (*Operation Mode*)
		JOG_POSITIVE, (*Jog positive state*)
		JOG_NEGATIVE, (*Jog Negative State*)
		IN_CUTTING_ZONE (*in Cutting zone state*)
		);
END_TYPE
```

#### Variables.var - Local variables
```iecst
(*********************************************************************************
 * Copyright: B&R Industrial Automation GmbH
 * Author:    kasliwals
 * Created:   December 11, 2023/10:45 AM
 *********************************************************************************)
(*Function Blocks*)
VAR
	iFb_MpAxisSlave : MpAxisBasic; (*MpAxis Function Block*)
	iFb_RegCapture : MC_BR_RegMarkCapture002; (*Reg Capture FB*)
	iFb_CamSeq : MpAxisCamSequencer; (*Cam Seq FB*)
	iFb_MpAxisBasic : MpAxisBasic; (*MpAxis Function Block*)
END_VAR
(*Axis Structures*)
VAR
	iAx_CamSeq : AxisCamSeqMain_Typ; (*Cam Seq Structure*)
	iCutterCtrl : AxisCtrl_typ; (*Cutter Ctrl Structure*)
END_VAR
(*CONSTANTS*)
VAR CONSTANT
	LOWER_CUT_POS : LREAL := 2653; (*Lower Limit of Cutting zone*)
	HOMING_OFFSET : LREAL := 1033; (*Homing Position*)
	UPPER_CUT_POS : LREAL := 3013; (*upper Limit of cutting zone*)
	START_VEL : REAL := 150; (*Start Velecity*)
	HOMING_VEL : REAL := 300; (*Homing Velocity*)
END_VAR
VAR
	ZERO : LREAL := 0; (*Zero number*)
	LIMIT_END : LREAL := 3599; (*Limit ENd*)
END_VAR
VAR CONSTANT
	LOWER_BUFER : LREAL := 2643; (*Lower Limit buffer*)
	UPPER_BUFFER : LREAL := 3014; (*Upper Limit buffer*)
END_VAR
(*Process Variables And Structures*)
VAR
	iVa_RegCaptureAdvPara : MC_BR_ADV_RM2_REF; (*Adv para for reg capture*)
	SlaveStateDual : AxisState_enum; (*Dual Cutter State*)
	SlaveStateSingle : AxisState_enum; (*Single Cutter State*)
	iVa_RegCaptureConfig : MC_BR_CFG_RM2_REF; (*Config Para for reg caoture*)
	sJogState : INT; (*Jog State*)
END_VAR
```

#### Mapping.st
```iecst
(*********************************************************************************
 * Copyright: B&R Industrial Automation GmbH
 * Author:    kasliwals
 * Created:   December 11, 2023/10:46 AM
* Description: Mapping Structure to Function blocks
* Version : 1.0.0.0
 *********************************************************************************)

ACTION Mapping:
	//Assising inputs of Master axis to function Block
	iFb_MpAxisBasic.MpLink       := ADR(gAxisMaster);
	iFb_MpAxisBasic.Enable       := gAx_Master.In.Enable;
	iFb_MpAxisBasic.ErrorReset   := gAx_Master.In.ErrorReset;
	iFb_MpAxisBasic.Parameters   := ADR(gAx_Master.In.Parameters);
	iFb_MpAxisBasic.Update       := gAx_Master.In.Update;
	iFb_MpAxisBasic.Axis         := ADR(gAxis01);
	iFb_MpAxisBasic.Power        := gAx_Master.In.Power;
	iFb_MpAxisBasic.Home         := gAx_Master.In.Home;
	iFb_MpAxisBasic.MoveVelocity := gAx_Master.In.MoveVelocity ;
	iFb_MpAxisBasic.MoveAbsolute := gAx_Master.In.MoveAbsolute;
	iFb_MpAxisBasic.MoveAdditive := gAx_Master.In.MoveAdditive  ;
	iFb_MpAxisBasic.Stop         := gAx_Master.In.Stop;
	iFb_MpAxisBasic.JogPositive  := gAx_Master.In.JogPositive;
	iFb_MpAxisBasic.JogNegative  := gAx_Master.In.JogNegative;
	iFb_MpAxisBasic.Autotune     := gAx_Master.In.Autotune;
	iFb_MpAxisBasic.Simulate     := gAx_Master.In.Simulate;
	iFb_MpAxisBasic.TorqueLimit  := gAx_Master.In.TorqueLimit;
	iFb_MpAxisBasic.ReleaseBrake := gAx_Master.In.ReleaseBrake;
	iFb_MpAxisBasic();
    //Assising Outputs of Master axis to function Block
	gAx_Master.Out.Active         := iFb_MpAxisBasic.Active;
	gAx_Master.Out.Error          := iFb_MpAxisBasic.Error;
	gAx_Master.Out.StatusID       := iFb_MpAxisBasic.StatusID;
	gAx_Master.Out.UpdateDone     := iFb_MpAxisBasic.UpdateDone;
	gAx_Master.Out.Position       := iFb_MpAxisBasic.Position;
	gAx_Master.Out.Velocity       := iFb_MpAxisBasic.Velocity;
	gAx_Master.Out.CommandBusy    := iFb_MpAxisBasic.CommandBusy;
	gAx_Master.Out.CommandAborted := iFb_MpAxisBasic.CommandAborted;
	gAx_Master.Out.PowerOn        := iFb_MpAxisBasic.PowerOn;
	gAx_Master.Out.IsHomed        := iFb_MpAxisBasic.IsHomed;
	gAx_Master.Out.InVelocity     := iFb_MpAxisBasic.InVelocity;
	gAx_Master.Out.InPosition     := iFb_MpAxisBasic.InPosition;
	gAx_Master.Out.MoveActive     := iFb_MpAxisBasic.MoveActive;
	gAx_Master.Out.Stopped        := iFb_MpAxisBasic.Stopped;
	gAx_Master.Out.TuningDone     := iFb_MpAxisBasic.TuningDone;
	gAx_Master.Out.Simulation     := iFb_MpAxisBasic.Simulation;
	gAx_Master.Out.TorqueLimited  := iFb_MpAxisBasic.TorqueLimited;
	gAx_Master.Out.BrakeReleased  := iFb_MpAxisBasic.BrakeReleased;
	gAx_Master.Out.Info           := iFb_MpAxisBasic.Info;

	//Assising inputs of Slave axis to function Block
	iFb_MpAxisSlave.MpLink       := ADR(gAxisSlave);
	iFb_MpAxisSlave.Enable       := gAx_Slave.In.Enable;
	iFb_MpAxisSlave.ErrorReset   := gAx_Slave.In.ErrorReset;
	iFb_MpAxisSlave.Parameters   := ADR(gAx_Slave.In.Parameters);
	iFb_MpAxisSlave.Update       := gAx_Slave.In.Update;
	iFb_MpAxisSlave.Axis         := ADR(gAxis02);
	iFb_MpAxisSlave.Power        := gAx_Slave.In.Power;
	iFb_MpAxisSlave.Home         := gAx_Slave.In.Home;
	iFb_MpAxisSlave.MoveVelocity := gAx_Slave.In.MoveVelocity ;
	iFb_MpAxisSlave.MoveAbsolute := gAx_Slave.In.MoveAbsolute;
	iFb_MpAxisSlave.MoveAdditive := gAx_Slave.In.MoveAdditive  ;
	iFb_MpAxisSlave.Stop         := gAx_Slave.In.Stop;
	iFb_MpAxisSlave.JogPositive  := gAx_Slave.In.JogPositive;
	iFb_MpAxisSlave.JogNegative  := gAx_Slave.In.JogNegative;
	iFb_MpAxisSlave.Autotune     := gAx_Slave.In.Autotune;
	iFb_MpAxisSlave.Simulate     := gAx_Slave.In.Simulate;
	iFb_MpAxisSlave.TorqueLimit  := gAx_Slave.In.TorqueLimit;
	iFb_MpAxisSlave.ReleaseBrake := gAx_Slave.In.ReleaseBrake;
	iFb_MpAxisSlave();
    //Assising Outputs of Slave axis to function Block
	gAx_Slave.Out.Active         := iFb_MpAxisSlave.Active;
	gAx_Slave.Out.Error          := iFb_MpAxisSlave.Error;
	gAx_Slave.Out.StatusID       := iFb_MpAxisSlave.StatusID;
	gAx_Slave.Out.UpdateDone     := iFb_MpAxisSlave.UpdateDone;
	gAx_Slave.Out.Position       := iFb_MpAxisSlave.Position;
	gAx_Slave.Out.Velocity       := iFb_MpAxisSlave.Velocity;
	gAx_Slave.Out.CommandBusy    := iFb_MpAxisSlave.CommandBusy;
	gAx_Slave.Out.CommandAborted := iFb_MpAxisSlave.CommandAborted;
	gAx_Slave.Out.PowerOn        := iFb_MpAxisSlave.PowerOn;
	gAx_Slave.Out.IsHomed        := iFb_MpAxisSlave.IsHomed;
	gAx_Slave.Out.InVelocity     := iFb_MpAxisSlave.InVelocity;
	gAx_Slave.Out.InPosition     := iFb_MpAxisSlave.InPosition;
	gAx_Slave.Out.MoveActive     := iFb_MpAxisSlave.MoveActive;
	gAx_Slave.Out.Stopped        := iFb_MpAxisSlave.Stopped;
	gAx_Slave.Out.TuningDone     := iFb_MpAxisSlave.TuningDone;
	gAx_Slave.Out.Simulation     := iFb_MpAxisSlave.Simulation;
	gAx_Slave.Out.TorqueLimited  := iFb_MpAxisSlave.TorqueLimited;
	gAx_Slave.Out.BrakeReleased  := iFb_MpAxisSlave.BrakeReleased;
	gAx_Slave.Out.Info           := iFb_MpAxisSlave.Info;

	//Assigning Output Structure to Axis Coupling Function Block
	iAx_CamSeq.Out.Active				:= iFb_CamSeq.Active;
	iAx_CamSeq.Out.Error				:= iFb_CamSeq.Error;
	iAx_CamSeq.Out.StatusID				:= iFb_CamSeq.StatusID;
	iAx_CamSeq.Out.UpdateDone			:= iFb_CamSeq.UpdateDone;
	iAx_CamSeq.Out.ActStIndex			:= iFb_CamSeq.ActualStateIndex;
	iAx_CamSeq.Out.ActStCamIndex		:= iFb_CamSeq.ActualStateCamIndex;
	iAx_CamSeq.Out.Standby				:= iFb_CamSeq.Standby;
	iAx_CamSeq.Out.InCompensation		:= iFb_CamSeq.InCompensation;
	iAx_CamSeq.Out.InSync				:= iFb_CamSeq.InSync;
	iAx_CamSeq.Out.Info					:= iFb_CamSeq.Info;

	//Assigning Input Structure to Axis Cam Sequencer Function Block
	iFb_CamSeq.MpLink					:= ADR(gAxisSlave);
	iFb_CamSeq.Enable					:= TRUE;
	iFb_CamSeq.ErrorReset				:= iAx_CamSeq.In.ErrorReset;
	iFb_CamSeq.Parameters				:= ADR(iAx_CamSeq.In.Parameters);
	iFb_CamSeq.Update					:= iAx_CamSeq.In.Update;
	iFb_CamSeq.MpLinkMaster				:= ADR(gAxisMaster);
	iFb_CamSeq.Signal1					:= iAx_CamSeq.In.Signal1;
	iFb_CamSeq.Signal2					:= iAx_CamSeq.In.Signal2;
	iFb_CamSeq.Signal3					:= iAx_CamSeq.In.Signal3;
	iFb_CamSeq.Signal4					:= iAx_CamSeq.In.Signal4;
	iFb_CamSeq.StartSequence			:= iAx_CamSeq.In.StartSequence;
	iFb_CamSeq.Continue					:= iAx_CamSeq.In.Continue;
	iFb_CamSeq.EndSequence				:= iAx_CamSeq.In.EndSequence;
	iFb_CamSeq();

END_ACTION
```

#### SingleCutter.st
```iecst
(*********************************************************************************
 * Copyright: B&R Industrial Automation GmbH
 * Author:    kasliwals
 * Created:   December 16, 2023/11:40 PM
* Description: Single Cutter Homingb Logic and jog Limits
* Version : 1.0.0.0
 *********************************************************************************)

ACTION  SingleCutter :
	CASE SlaveStateSingle OF
		WAIT :
			IF gAx_Slave.Out.Active AND iCutterCtrl.Cmd.Start THEN
				SlaveStateSingle := POWER_ON;
			END_IF
		ACTIVE :
			IF gAx_Slave.Out.Position >= LOWER_CUT_POS AND gAx_Master.Out.Position <= UPPER_CUT_POS THEN
				gAx_Slave.In.Power := FALSE;
			ELSE
				SlaveStateSingle := POWER_ON;
			END_IF

		POWER_ON :
			IF gAx_Slave.Out.Info.ReadyToPowerOn  AND iCutterCtrl.Cmd.AutoMode  THEN
				gAx_Slave.In.Power := TRUE;
			END_IF
			IF gAx_Slave.Out.PowerOn AND gAx_Slave.Out.Position < LOWER_CUT_POS THEN
				SlaveStateSingle := NEGATIVE_HOMING_MODE;
			END_IF
			IF gAx_Slave.Out.PowerOn AND gAx_Slave.Out.Position > UPPER_CUT_POS THEN
				SlaveStateSingle := POSITIVE_HOMING_MODE;
			END_IF

		NEGATIVE_HOMING_MODE :
			gAx_Slave.In.Parameters.Home.Mode := mpAXIS_HOME_MODE_REF_PULSE;
			gAx_Slave.In.Parameters.Home.HomingDirection := mpAXIS_HOME_DIR_NEGATIVE;
			gAx_Slave.In.Parameters.Home.SensorOffset := HOMING_OFFSET;
			gAx_Slave.In.Parameters.Home.HomingVelocity := HOMING_VEL;
			gAx_Slave.In.Parameters.Home.StartVelocity := START_VEL;
			gAx_Slave.In.Update := TRUE;
			IF gAx_Slave.Out.UpdateDone THEN
				gAx_Slave.In.Update := FALSE;
				gAx_Slave.In.Home := TRUE;
				SlaveStateSingle := HOMING;
			END_IF
		POSITIVE_HOMING_MODE :
			gAx_Slave.In.Parameters.Home.Mode := mpAXIS_HOME_MODE_REF_PULSE;
			gAx_Slave.In.Parameters.Home.HomingDirection := mpAXIS_HOME_DIR_POSITIVE;
			gAx_Slave.In.Parameters.Home.SensorOffset := HOMING_OFFSET;
			gAx_Slave.In.Parameters.Home.HomingVelocity := HOMING_VEL;
			gAx_Slave.In.Parameters.Home.StartVelocity := START_VEL;

			gAx_Slave.In.Update := TRUE;
			IF gAx_Slave.Out.UpdateDone THEN
				gAx_Slave.In.Update := FALSE;
				gAx_Slave.In.Home := TRUE;
				SlaveStateSingle := HOMING;
			END_IF

		HOMING :
			IF gAx_Slave.Out.IsHomed THEN
				gAx_Slave.In.Home := FALSE;
				IF iCutterCtrl.Cmd.AutoMode THEN
					SlaveStateSingle := AUTO_MODE;
				ELSE
					SlaveStateSingle := OPERATION;
				END_IF

			END_IF

		AUTO_MODE :
			IF iCutterCtrl.Cmd.Start = FALSE THEN
				SlaveStateSingle := WAIT;
			END_IF

		OPERATION :
			IF iCutterCtrl.Cmd.JogFwd THEN
				SlaveStateSingle := JOG_POSITIVE;
			END_IF
			IF iCutterCtrl.Cmd.JogBack THEN
				SlaveStateSingle := JOG_NEGATIVE;
			END_IF
			IF iCutterCtrl.Cmd.Start = FALSE THEN
				SlaveStateSingle := WAIT;
			END_IF

		JOG_POSITIVE :
			IF NOT iCutterCtrl.Cmd.JogFwd OR gAx_Slave.Out.Position = LOWER_BUFER  THEN
				gAx_Slave.In.JogPositive := FALSE;
				SlaveStateSingle := OPERATION;
			ELSE
				gAx_Slave.In.JogPositive := TRUE;
			END_IF
			IF gAx_Slave.Out.Position = LOWER_BUFER THEN
				iCutterCtrl.Cmd.JogFwd := FALSE;
			END_IF

		JOG_NEGATIVE :
			IF NOT iCutterCtrl.Cmd.JogBack OR gAx_Slave.Out.Position = UPPER_BUFFER  THEN
				gAx_Slave.In.JogNegative := FALSE;
				SlaveStateSingle := OPERATION;
			ELSE
				gAx_Slave.In.JogNegative := TRUE;
			END_IF
			IF gAx_Slave.Out.Position = UPPER_BUFFER THEN
				iCutterCtrl.Cmd.JogBack := FALSE;
			END_IF

		IN_CUTTING_ZONE :
			gAx_Slave.In.Power := FALSE;
			IF (gAx_Slave.Out.Position < LOWER_CUT_POS OR gAx_Slave.Out.Position >UPPER_CUT_POS) AND gAx_Slave.Out.IsHomed THEN
				gAx_Slave.In.Power := TRUE;
				SlaveStateSingle := OPERATION;
			ELSIF  (gAx_Slave.Out.Position < LOWER_CUT_POS OR gAx_Slave.Out.Position >UPPER_CUT_POS) AND NOT gAx_Slave.Out.IsHomed THEN
				SlaveStateSingle := POWER_ON;
			END_IF

	END_CASE

	CASE sJogState OF
		0:
			IF gAx_Slave.In.JogNegative = TRUE THEN
				sJogState	:= 10;
			END_IF;
			IF (gAx_Slave.In.JogPositive = TRUE) THEN
				sJogState	:= 20;
			END_IF;
		5:
			gAx_Slave.In.JogPositive	:= TRUE;
			gAx_Slave.In.JogNegative	:= TRUE;
			sJogState		:= 0;

		10:
			IF (gAx_Slave.Out.CommandAborted = TRUE) THEN
				sJogState					:= 5;
				gAx_Slave.In.JogNegative	:= FALSE;
			END_IF;

			IF (gAx_Slave.Out.Position > UPPER_CUT_POS)THEN
				gAx_Slave.In.Parameters.Jog.LowerLimit	:= UPPER_BUFFER;
				gAx_Slave.In.Parameters.Jog.UpperLimit	:= LIMIT_END;
				gAx_Slave.In.Update					:= TRUE;
				sJogState								:= 30;
			END_IF;
		20:
			IF (gAx_Slave.Out.CommandAborted = TRUE) THEN
				sJogState					:= 5;
				gAx_Slave.In.JogPositive	:= FALSE;
			END_IF;

			IF (gAx_Slave.Out.Position < LOWER_CUT_POS)THEN
				gAx_Slave.In.Parameters.Jog.LowerLimit	:=ZERO;
				gAx_Slave.In.Parameters.Jog.UpperLimit	:= LOWER_BUFER;
				gAx_Slave.In.Update					:= TRUE;
				sJogState								:= 30;
			END_IF;
		30:
			IF gAx_Slave.Out.UpdateDone = TRUE THEN
				gAx_Slave.In.Update					:= FALSE;
			END_IF;
			IF gAx_Slave.In.JogNegative = TRUE AND gAx_Slave.Out.Position <ZERO AND gAx_Slave.Out.Position > UPPER_CUT_POS THEN
				sJogState	:= 10;
			END_IF;
			IF (gAx_Slave.In.JogPositive = TRUE) AND gAx_Slave.Out.Position > ZERO AND gAx_Slave.Out.Position < LOWER_CUT_POS  THEN
				sJogState	:= 20;
			END_IF;
			IF ((gAx_Slave.Out.Position = UPPER_BUFFER) OR (gAx_Slave.Out.Position =LOWER_BUFER )) THEN
				gAx_Slave.In.JogNegative			:= FALSE;
				gAx_Slave.In.JogPositive			:= FALSE;
				sJogState							:= 40;
			END_IF;
		40:

			gAx_Slave.In.Parameters.Jog.LowerLimit	:= ZERO;
			gAx_Slave.In.Parameters.Jog.UpperLimit	:= ZERO;
			gAx_Slave.In.Update					:= TRUE;
			IF gAx_Slave.Out.UpdateDone = TRUE THEN
				gAx_Slave.In.Update				:= FALSE;
				sJogState							:= 0;
			END_IF;
	END_CASE;

//	IF gAx_Slave.Out.Position >=LOWER_CUT_POS AND gAx_Slave.Out.Position <=UPPER_CUT_POS THEN
//		iCutterCtrl.Status.JogNegReady := FALSE;
//		iCutterCtrl.Status.JogPosReady := FALSE;
//		SlaveStateSingle := IN_CUTTING_ZONE;
//
//	END_IF

END_ACTION
```

#### DualCutter.st
```iecst
(*********************************************************************************
 * Copyright: B&R Industrial Automation GmbH
 * Author:    kasliwals
 * Created:   December 16, 2023/11:41 PM
* Description: Dual Cutter Homing Logic and jog limits
* Version : 1.0.0.0
 *********************************************************************************)

ACTION DualCutter:
	CASE SlaveStateDual OF
		WAIT :
			IF gAx_Slave.Out.Active THEN
				SlaveStateDual := ACTIVE ;
			END_IF

		ACTIVE :
			IF gAx_Slave.Out.Info.ReadyToPowerOn THEN
				gAx_Slave.In.Power := TRUE;
			END_IF
			IF gAx_Slave.Out.PowerOn AND gAx_Slave.Out.Position > 3013 THEN
				SlaveStateDual := POSITIVE_HOMING_MODE;
			END_IF
			IF gAx_Slave.Out.PowerOn AND gAx_Slave.Out.Position > 142 AND gAx_Slave.Out.Position < 853 THEN
				SlaveStateDual := NEGATIVE_HOMING_MODE;
			END_IF

		NEGATIVE_HOMING_MODE :
			gAx_Slave.In.Parameters.Home.Mode := mpAXIS_HOME_MODE_REF_PULSE;
			gAx_Slave.In.Parameters.Home.HomingDirection := mpAXIS_HOME_DIR_NEGATIVE;
			gAx_Slave.In.Parameters.Home.HomingVelocity := 300;
			gAx_Slave.In.Parameters.Position := 142;
			gAx_Slave.In.Parameters.Velocity := 300;
			gAx_Slave.In.Update := TRUE;
			IF gAx_Slave.Out.UpdateDone THEN
				gAx_Slave.In.Update := FALSE;
				gAx_Slave.In.Home := TRUE;
				SlaveStateDual := HOMING;
			END_IF
		POSITIVE_HOMING_MODE :
			gAx_Slave.In.Parameters.Home.Mode := mpAXIS_HOME_MODE_REF_PULSE;
			gAx_Slave.In.Parameters.Home.HomingDirection := mpAXIS_HOME_DIR_POSITIVE;
			gAx_Slave.In.Parameters.Home.HomingVelocity := 300;
			gAx_Slave.In.Parameters.Position := 142;
			gAx_Slave.In.Parameters.Velocity := 300;
			gAx_Slave.In.Update := TRUE;
			IF gAx_Slave.Out.UpdateDone THEN
				gAx_Slave.In.Update := FALSE;
				gAx_Slave.In.Home := TRUE;
				SlaveStateDual := HOMING;
			END_IF

		HOMING :
			IF gAx_Slave.Out.IsHomed THEN
				gAx_Slave.In.Home := FALSE;
				gAx_Slave.In.MoveAbsolute := TRUE;
			END_IF
			IF gAx_Slave.Out.InPosition THEN
				gAx_Slave.In.MoveAbsolute := FALSE;
				SlaveStateDual := OPERATION;
			END_IF

		OPERATION :
	END_CASE

END_ACTION
```

#### CamAuto.st
```iecst
(*********************************************************************************
 * Copyright: B&R Industrial Automation GmbH
 * Author:    kasliwals
 * Created:   December 16, 2023/11:41 PM
* Description: Cam Automat for Single Cutter and Dual Cutter
* Version : 1.0.0.0
 *********************************************************************************)

ACTION SingleCam:
	iAx_CamSeq.In.Parameters.Configuration.Master := ADR(gAxis01); // Not Mplink Axis Address
	iAx_CamSeq.In.Parameters.Configuration.MasterParID := ACP10PAR_PCTRL_S_ACT; //412 parid -
	(** STATE 0 - Event 1 - WAIT FOR TRIGGER **)

	iAx_CamSeq.In.Parameters.Configuration.State[0].Event[0].Type := ncTRIGGER1; //Trigger
	iAx_CamSeq.In.Parameters.Configuration.State[0].Event[0].Attribute := ncAT_ONCE; //Reaction
	iAx_CamSeq.In.Parameters.Configuration.State[0].Event[0].NextState := 3; //Next State
	(** STATE 1 - WAIT FOR TRIGGER **)

	iAx_CamSeq.In.Parameters.Configuration.State[1].CamProfileIndex := 16#FFFE;
	iAx_CamSeq.In.Parameters.Configuration.State[1].MasterFactor := 300 ; //Master Dist.
	iAx_CamSeq.In.Parameters.Configuration.State[1].SlaveFactor := -400; //Slave Dist.

	iAx_CamSeq.In.Parameters.Configuration.State[1].CompMode := ncONLYCOMP;
	iAx_CamSeq.In.Parameters.Configuration.State[1].MasterCompDistance := 400; //Master Dist.
	iAx_CamSeq.In.Parameters.Configuration.State[1].SlaveCompDistance := -3200; //Slave Dist.

	iAx_CamSeq.In.Parameters.Configuration.State[1].Event[0].Type := ncST_END; //Trigger
	iAx_CamSeq.In.Parameters.Configuration.State[1].Event[0].Attribute := ncST_END; //Reaction
	iAx_CamSeq.In.Parameters.Configuration.State[1].Event[0].NextState := 2; //Next State

	iAx_CamSeq.In.Parameters.Configuration.State[2].CamProfileIndex := 16#FFFF;
	iAx_CamSeq.In.Parameters.Configuration.State[2].MasterFactor := 300; //Master Dist.
	iAx_CamSeq.In.Parameters.Configuration.State[2].SlaveFactor := -400; //Slave Dist.

	iAx_CamSeq.In.Parameters.Configuration.State[2].Event[0].Type := ncST_END; //Trigger
	iAx_CamSeq.In.Parameters.Configuration.State[2].Event[0].Attribute := ncST_END; //Reaction
	iAx_CamSeq.In.Parameters.Configuration.State[2].Event[0].NextState := 1; //Next State

	//ONLY FOR FIRST PRINT MARK
	iAx_CamSeq.In.Parameters.Configuration.State[3].CamProfileIndex := 16#FFFE;
	iAx_CamSeq.In.Parameters.Configuration.State[3].MasterFactor := 300; //Master Dist.
	iAx_CamSeq.In.Parameters.Configuration.State[3].SlaveFactor := -400; //Slave Dist.

	iAx_CamSeq.In.Parameters.Configuration.State[3].CompMode := ncONLYCOMP;
	iAx_CamSeq.In.Parameters.Configuration.State[3].MasterCompDistance := 1650; //Master Dist.
	iAx_CamSeq.In.Parameters.Configuration.State[3].SlaveCompDistance := -1580; //Slave Dist.

	iAx_CamSeq.In.Parameters.Configuration.State[3].Event[0].Type :=ncST_END; //Trigger
	iAx_CamSeq.In.Parameters.Configuration.State[3].Event[0].Attribute := ncST_END; //Reaction
	iAx_CamSeq.In.Parameters.Configuration.State[3].Event[0].NextState := 2; //Next State

END_ACTION

ACTION DualCutterCamAuto :
	iAx_CamSeq.In.Parameters.Configuration.Master := ADR(gAxis01); // Not Mplink Axis Address
	iAx_CamSeq.In.Parameters.Configuration.MasterParID := ACP10PAR_PCTRL_S_ACT; //412 parid -
	(** STATE 0 - Event 1 - WAIT FOR TRIGGER **)

	iAx_CamSeq.In.Parameters.Configuration.State[0].Event[0].Type := ncTRIGGER1; //Trigger
	iAx_CamSeq.In.Parameters.Configuration.State[0].Event[0].Attribute := ncAT_ONCE; //Reaction
	iAx_CamSeq.In.Parameters.Configuration.State[0].Event[0].NextState := 3; //Next State
	(** STATE 1 - WAIT FOR TRIGGER **)

	iAx_CamSeq.In.Parameters.Configuration.State[1].CamProfileIndex := 16#FFFE;
	iAx_CamSeq.In.Parameters.Configuration.State[1].MasterFactor := 300 ; //Master Dist.
	iAx_CamSeq.In.Parameters.Configuration.State[1].SlaveFactor := -400; //Slave Dist.

	iAx_CamSeq.In.Parameters.Configuration.State[1].CompMode := ncONLYCOMP;
	iAx_CamSeq.In.Parameters.Configuration.State[1].MasterCompDistance := 400; //Master Dist.
	iAx_CamSeq.In.Parameters.Configuration.State[1].SlaveCompDistance := -1400; //Slave Dist.

	iAx_CamSeq.In.Parameters.Configuration.State[1].Event[0].Type := ncST_END; //Trigger
	iAx_CamSeq.In.Parameters.Configuration.State[1].Event[0].Attribute := ncST_END; //Reaction
	iAx_CamSeq.In.Parameters.Configuration.State[1].Event[0].NextState := 2; //Next State

	iAx_CamSeq.In.Parameters.Configuration.State[2].CamProfileIndex := 16#FFFF;
	iAx_CamSeq.In.Parameters.Configuration.State[2].MasterFactor := 300; //Master Dist.
	iAx_CamSeq.In.Parameters.Configuration.State[2].SlaveFactor := -400; //Slave Dist.

	iAx_CamSeq.In.Parameters.Configuration.State[2].Event[0].Type := ncST_END; //Trigger
	iAx_CamSeq.In.Parameters.Configuration.State[2].Event[0].Attribute := ncST_END; //Reaction
	iAx_CamSeq.In.Parameters.Configuration.State[2].Event[0].NextState := 1; //Next State

	//ONLY FOR FIRST PRINT MARK
	iAx_CamSeq.In.Parameters.Configuration.State[3].CamProfileIndex := 16#FFFE;
	iAx_CamSeq.In.Parameters.Configuration.State[3].MasterFactor := 300; //Master Dist.
	iAx_CamSeq.In.Parameters.Configuration.State[3].SlaveFactor := -400; //Slave Dist.

	iAx_CamSeq.In.Parameters.Configuration.State[3].CompMode := ncONLYCOMP;
	iAx_CamSeq.In.Parameters.Configuration.State[3].MasterCompDistance := 1650; //Master Dist.
	iAx_CamSeq.In.Parameters.Configuration.State[3].SlaveCompDistance := -700; //Slave Dist.

	iAx_CamSeq.In.Parameters.Configuration.State[3].Event[0].Type :=ncST_END; //Trigger
	iAx_CamSeq.In.Parameters.Configuration.State[3].Event[0].Attribute := ncST_END; //Reaction
	iAx_CamSeq.In.Parameters.Configuration.State[3].Event[0].NextState := 2; //Next State
	END_ACTION
```

#### regCapture.st
```iecst
(*********************************************************************************
 * Copyright: B&R Industrial Automation GmbH
 * Author:    kasliwals
 * Created:   December 16, 2023/11:41 PM
* Description: Reg Capture implementation
* Version : 1.0.0.0
 *********************************************************************************)

ACTION RegCapture:
	iFb_RegCapture.Axis := ADR(gAxis02);
	iFb_RegCapture.Master := ADR(gAxis01);
	iFb_RegCapture.AdvancedParameters := iVa_RegCaptureAdvPara;
	iFb_RegCapture.InitData := TRUE;
	iFb_RegCapture.SearchRM := TRUE;
	iFb_RegCapture.Configuration := iVa_RegCaptureConfig;
	iFb_RegCapture.CutPosition := REAL_TO_DINT(iVa_RegCaptureConfig.ProductLength);
	iFb_RegCapture.Enable := iAx_CamSeq.Out.InSync;
	IF gAx_Slave.Out.Info.PLCopenState = mpAXIS_SYNCHRONIZED_MOTION THEN
		iFb_RegCapture();
	END_IF
END_ACTION
```

#### SingleCutterCamAuto.st - not listed in the package file held
```iecst
ACTION SingleCam:
	iAx_CamSeq.In.Parameters.Configuration.Master := ADR(gAxis01); // Not Mplink Axis Address
	iAx_CamSeq.In.Parameters.Configuration.MasterParID := ACP10PAR_PCTRL_S_ACT; //412 parid -
	(** STATE 0 - Event 1 - WAIT FOR TRIGGER **)

	iAx_CamSeq.In.Parameters.Configuration.State[0].Event[0].Type := ncTRIGGER1; //Trigger
	iAx_CamSeq.In.Parameters.Configuration.State[0].Event[0].Attribute := ncAT_ONCE; //Reaction
	iAx_CamSeq.In.Parameters.Configuration.State[0].Event[0].NextState := 3; //Next State
	(** STATE 1 - WAIT FOR TRIGGER **)

	iAx_CamSeq.In.Parameters.Configuration.State[1].CamProfileIndex := 16#FFFE;
	iAx_CamSeq.In.Parameters.Configuration.State[1].MasterFactor := 300 ; //Master Dist.
	iAx_CamSeq.In.Parameters.Configuration.State[1].SlaveFactor := -400; //Slave Dist.

	iAx_CamSeq.In.Parameters.Configuration.State[1].CompMode := ncONLYCOMP;
	iAx_CamSeq.In.Parameters.Configuration.State[1].MasterCompDistance := 400; //Master Dist.
	iAx_CamSeq.In.Parameters.Configuration.State[1].SlaveCompDistance := -3200; //Slave Dist.

	iAx_CamSeq.In.Parameters.Configuration.State[1].Event[0].Type := ncST_END; //Trigger
	iAx_CamSeq.In.Parameters.Configuration.State[1].Event[0].Attribute := ncST_END; //Reaction
	iAx_CamSeq.In.Parameters.Configuration.State[1].Event[0].NextState := 2; //Next State

	iAx_CamSeq.In.Parameters.Configuration.State[2].CamProfileIndex := 16#FFFF;
	iAx_CamSeq.In.Parameters.Configuration.State[2].MasterFactor := 300; //Master Dist.
	iAx_CamSeq.In.Parameters.Configuration.State[2].SlaveFactor := -400; //Slave Dist.

	iAx_CamSeq.In.Parameters.Configuration.State[2].Event[0].Type := ncST_END; //Trigger
	iAx_CamSeq.In.Parameters.Configuration.State[2].Event[0].Attribute := ncST_END; //Reaction
	iAx_CamSeq.In.Parameters.Configuration.State[2].Event[0].NextState := 1; //Next State

	//ONLY FOR FIRST PRINT MARK
	iAx_CamSeq.In.Parameters.Configuration.State[3].CamProfileIndex := 16#FFFE;
	iAx_CamSeq.In.Parameters.Configuration.State[3].MasterFactor := 300; //Master Dist.
	iAx_CamSeq.In.Parameters.Configuration.State[3].SlaveFactor := -400; //Slave Dist.

	iAx_CamSeq.In.Parameters.Configuration.State[3].CompMode := ncONLYCOMP;
	iAx_CamSeq.In.Parameters.Configuration.State[3].MasterCompDistance := 1650; //Master Dist.
	iAx_CamSeq.In.Parameters.Configuration.State[3].SlaveCompDistance := -1580; //Slave Dist.

	iAx_CamSeq.In.Parameters.Configuration.State[3].Event[0].Type :=ncST_END; //Trigger
	iAx_CamSeq.In.Parameters.Configuration.State[3].Event[0].Attribute := ncST_END; //Reaction
	iAx_CamSeq.In.Parameters.Configuration.State[3].Event[0].NextState := 2; //Next State

END_ACTION
```

### AxisTyp.typ - Axis global structures
```iecst
(*********************************************************************************
 * Copyright: B&R Industrial Automation GmbH
 * Author:    kasliwals
 * Created:   December 11, 2023/10:46 AM
 *********************************************************************************)
(*Cam Sequencxe Structure*)

TYPE
	AxisCamSeqInput_Typ : 	STRUCT  (*Cam sequence Input structure type*)
		ErrorReset : BOOL; (*Resets function block errors*) (* *) (*#PAR#;*)
		Parameters : MpAxisCamSequencerParType; (*Function block parameters*) (* *) (*#PAR#;*)
		Update : BOOL; (*Update command for the parameters*) (* *) (*#PAR#;*)
		Signal1 : BOOL; (*Starts a cam profile used by the slave to follow the master*) (* *) (*#CMD#;*)
		Signal2 : BOOL; (*Begins to undo all shifts made*) (* *) (*#CMD#OPT#;*)
		Signal3 : BOOL; (*Starts a phase shift to the slave position (offset)*) (* *) (*#CMD#OPT#;*)
		Signal4 : BOOL; (*Starts a phase shift to the master position with which the slave is working (phase); the master remains unaffected*) (* *) (*#CMD#OPT#;*)
		StartSequence : BOOL; (*Starts a phase shift to the master position with which the slave is working (phase); the master remains unaffected*) (* *) (*#CMD#OPT#;*)
		Continue : BOOL; (*Starts a phase shift to the master position with which the slave is working (phase); the master remains unaffected*) (* *) (*#CMD#OPT#;*)
		EndSequence : BOOL; (*Starts a phase shift to the master position with which the slave is working (phase); the master remains unaffected*) (* *) (*#CMD#OPT#;*)
	END_STRUCT;
	AxisCamSeqOutput_Typ : 	STRUCT  (*Cam sequence Output structure type*)
		Active : BOOL; (*Indicates whether the function block is active*) (* *) (*#PAR#;*)
		Error : BOOL; (*Indicates that the function block is in an error state or a command was not executed correctly*) (* *) (*#PAR#;*)
		UpdateDone : BOOL; (*Parameter update completed*) (* *) (*#PAR#;*)
		ActStIndex : USINT; (*Function block currently executing command*) (* *) (*#CMD#OPT#;*)
		ActStCamIndex : UINT; (*Function block interrupted while executing a command*) (* *) (*#CMD#OPT#;*)
		StatusID : DINT; (*Status information about the function block*) (* *) (*#PAR#;*)
		Info : MpAxisCamSequencerInfoType; (*Additional information about the component*) (* *) (*#CMD#;*)
		Standby : BOOL; (*Standby Output var for Cam Sequence*)
		InCompensation : BOOL; (*Compensation Output var for Cam Sequence*)
		InSync : BOOL; (*Sync Output var for Cam Sequence*)
	END_STRUCT;
	AxisCamSeqMain_Typ : 	STRUCT  (*Cam Sequence Main structure type*)
		In : AxisCamSeqInput_Typ; (*Variable to bind with input structure*)
		Out : AxisCamSeqOutput_Typ; (*Variable to bind with output structure*)
	END_STRUCT;
END_TYPE

(*Axis basic Structure*)

TYPE
	AxisBasicIn_type : 	STRUCT  (*Axis Input Structure *)
		ErrorReset : BOOL; (*Resets function block errors*) (* *) (*#PAR#;*)
		Parameters : MpAxisBasicParType; (*Function block parameters*) (* *) (*#PAR#;*)
		Update : BOOL; (*Updates the parameters*) (* *) (*#PAR#;*)
		Power : BOOL; (*Level-sensitive command for turning an axis on/off. In the event of an error, a new rising edge is required to restart the axis*) (* *) (*#CMD#;*)
		Home : BOOL; (*Command for homing the axis*) (* *) (*#CMD#;*)
		MoveVelocity : BOOL; (*Starts a constant movement with a defined velocity*) (* *) (*#CMD#;*)
		MoveAbsolute : BOOL; (*Starts an absolute movement*) (* *) (*#CMD#;*)
		MoveAdditive : BOOL; (*Starts a relative movement*) (* *) (*#CMD#;*)
		Stop : BOOL; (*Stops the axis*) (* *) (*#CMD#;*)
		JogPositive : BOOL; (*Movement in the positive direction. Stops automatically at the software limit position*) (* *) (*#CMD#OPT#;*)
		JogNegative : BOOL; (*Movement in the negative direction. Stops automatically at the software limit position*) (* *) (*#CMD#OPT#;*)
		Autotune : BOOL; (*Starts autotuning*) (* *) (*#CMD#OPT#;*)
		Simulate : BOOL; (*Enables motor simulation*) (* *) (*#CMD#OPT#;*)
		TorqueLimit : BOOL; (*Enables torque limiting*) (* *) (*#CMD#OPT#;*)
		ReleaseBrake : BOOL; (*Locks or unlocks the holding brake (only when the axis is switched off)*) (* *) (*#CMD#OPT#;*)
		Enable : BOOL;
	END_STRUCT;
	AxisBasicOut_type : 	STRUCT  (*Axis OutPut Structure*)
		Active : BOOL; (*Indicates whether the function block is active*) (* *) (*#PAR#;*)
		Error : BOOL; (*Indicates that the function block is in an error state or a command was not executed correctly*) (* *) (*#PAR#;*)
		StatusID : DINT; (*Status information about the function block*) (* *) (*#PAR#;*)
		UpdateDone : BOOL; (*Parameter update completed*) (* *) (*#PAR#;*)
		Position : LREAL; (*Current position of the axis [units]*) (* *) (*#CYC#;*)
		Velocity : REAL; (*Current position of the axis [units/s]*) (* *) (*#CYC#;*)
		CommandBusy : BOOL; (*Function block currently executing command*) (* *) (*#CMD#OPT#;*)
		CommandAborted : BOOL; (*Function block interrupted while executing a command*) (* *) (*#CMD#OPT#;*)
		PowerOn : BOOL; (*Switches on the axis*) (* *) (*#CMD#;*)
		IsHomed : BOOL; (*Homes the axis*) (* *) (*#CMD#;*)
		InVelocity : BOOL; (*Axis running with defined velocity*) (* *) (*#CMD#;*)
		InPosition : BOOL; (*Axis reached the desired position*) (* *) (*#CMD#;*)
		MoveActive : BOOL; (*Movement active*) (* *) (*#CMD#;*)
		Stopped : BOOL; (*Axis stopped*) (* *) (*#CMD#;*)
		TuningDone : BOOL; (*Autotuning completed successfully*) (* *) (*#CMD#OPT#;*)
		Simulation : BOOL; (*Motor simulation active*) (* *) (*#CMD#OPT#;*)
		TorqueLimited : BOOL; (*Torque limiting function active*) (* *) (*#CMD#OPT#;*)
		BrakeReleased : BOOL; (*Holding brake manually released*) (* *) (*#CMD#OPT#;*)
		Info : MpAxisBasicInfoType; (*Additional information about the component*) (* *) (*#CMD#;*)
	END_STRUCT;
	AxisBasic_type : 	STRUCT  (*Axis Main Structure type*)
		In : AxisBasicIn_type;
		Out : AxisBasicOut_type;
	END_STRUCT;
	AxisCtrl_typ : 	STRUCT  (*Axis Ctrl Struture*)
		Cmd : AxisCmd_typ; (*Axis Ctrl CMd type*)
		Para : AxisPara_typ; (*Axis para type*)
		Status : AxisStatus_typ; (*Axis Status Type*)
	END_STRUCT;
	AxisCmd_typ : 	STRUCT  (*Axis Ctrl CMd type*)
		Start : BOOL; (*Start Cmd*)
		Stop : BOOL; (*Stop cmd*)
		PrintMark : BOOL; (*Print mark detection bit*)
		ErrorReset : BOOL; (*Error reset*)
		AutoMode : BOOL; (*AutoMode*)
		JogFwd : BOOL; (*Jog fwd cmd*)
		JogBack : BOOL; (*jog BAck cmd*)
		Home : BOOL; (*home Cmd*)
	END_STRUCT;
	AxisPara_typ : 	STRUCT
		Speed : UINT; (*Axis Speed*)
	END_STRUCT;
	AxisStatus_typ : 	STRUCT  (*Axis Status*)
		JogNegReady : BOOL; (*Axis jog neg ready status*)
		JogPosReady : BOOL; (*axis jog pos ready Statsus*)
	END_STRUCT;
END_TYPE
```

### Program Logical/Source/AxisConf/ConvCtrl (IEC) - Conv Ctrl Logic

#### Types.typ
```iecst
(*********************************************************************************
 * Copyright: B&R Industrial Automation GmbH
 * Author:    kasliwals
 * Created:   December 16, 2023/11:44 PM
 *********************************************************************************)

TYPE
	MasterAxisState_enum :
		( (*Master Axis States*)
		WAIT, (*Wait State*)
		ACTIVE, (*ACtive State*)
		POWER_ON, (*Power On State*)
		HOME, (*HOMING State*)
		READY_TO_START, (*Ready to Start State*)
		MODE_CHANGE, (*Mode change state*)
		MANUAL, (*Manual state*)
		AUTOMATIC, (*Auto mode state*)
		JOG_POSITIVE, (*Jog Positive State*)
		JOG_NEGATIVE, (*Jog Negative State*)
		STOP (*Stop State*)
		);
END_TYPE
```

#### Variables.var
```iecst
(*********************************************************************************
 * Copyright: B&R Industrial Automation GmbH
 * Author:    kasliwals
 * Created:   December 16, 2023/11:45 PM
 *********************************************************************************)
(*Process Variables*)
VAR
	MasterStep : MasterAxisState_enum; (*Master state Variables*)
	iConvCtrl : AxisCtrl_typ; (*Conv Ctrl Structure*)
	iVa_SetMasterInputs : MC_BR_SetHardwareInputs; (*Set hardware FB*)
	iVa_RecPrintPosition : LREAL; (*Rec Print Pos Variable*)
END_VAR
(*Constants*)
VAR CONSTANT
	PRINT_MARK_LIMIT : LREAL := 300; (*Print maark limit*)
	MM_TO_UDINT : LREAL := 0.0; (*MM to udint conversion*)
	K_ZERO : LREAL := 0.0; (*Zero number*)
END_VAR
```

#### Main.st
```iecst
(*********************************************************************************
 * Copyright: B&R Industrial Automation GmbH
 * Author:    kasliwals
 * Created:   December 16, 2023/11:44 PM
* Description: Conv Homing and jog logic
* Version : 1.0.0.0
 *********************************************************************************)

PROGRAM _INIT
	(* Insert code here *)
	gAx_Master.In.Parameters.Jog.Acceleration := 480000;
	gAx_Master.In.Parameters.Jog.Deceleration := 4800000;
	gAx_Master.In.Parameters.Jog.Velocity := 45;
	gAx_Master.In.Parameters.Home.Mode := mpAXIS_HOME_MODE_ABS_SWITCH;
	gAx_Master.In.Parameters.Home.StartVelocity := 200;
	gAx_Master.In.Parameters.Home.HomingDirection := mpAXIS_HOME_DIR_NEGATIVE;

END_PROGRAM

PROGRAM _CYCLIC
	CASE MasterStep OF
		WAIT :
			IF gAx_Master.Out.Active AND iConvCtrl.Cmd.Start THEN
				MasterStep := ACTIVE;
			END_IF

		ACTIVE :
			IF gAx_Master.Out.Info.ReadyToPowerOn AND iConvCtrl.Cmd.AutoMode THEN
				gAx_Master.In.Power := TRUE;
			END_IF
			IF gAx_Master.Out.PowerOn THEN
				MasterStep := HOME;
			END_IF

		HOME :

				gAx_Master.In.Home := TRUE;

			IF gAx_Master.Out.IsHomed THEN
				gAx_Master.In.Home := FALSE;
				IF iConvCtrl.Cmd.AutoMode THEN
					MasterStep := AUTOMATIC;
				ELSE
					MasterStep := MANUAL;
				END_IF

			END_IF

		AUTOMATIC :
			IF iConvCtrl.Cmd.Start = FALSE THEN

				MasterStep := WAIT;
			END_IF

		MANUAL :
			IF iConvCtrl.Cmd.JogFwd THEN
				MasterStep := JOG_POSITIVE;
			END_IF
			IF iConvCtrl.Cmd.JogBack THEN
				MasterStep := JOG_NEGATIVE;
			END_IF
			iVa_RecPrintPosition := K_ZERO;
			IF iConvCtrl.Cmd.Start = FALSE THEN
				MasterStep := WAIT;
				gAx_Master.In.Power := FALSE;
			END_IF

		JOG_POSITIVE :
			gAx_Master.In.JogPositive := TRUE;
			IF NOT iConvCtrl.Cmd.JogFwd THEN
				gAx_Master.In.JogPositive := FALSE;
				MasterStep := MANUAL;
			END_IF

		JOG_NEGATIVE :
			gAx_Master.In.JogNegative := TRUE;
			IF (gAx_Master.In.JogNegative  AND EDGENEG(iConvCtrl.Cmd.PrintMark)) OR
				(EDGEPOS(gAx_Master.In.JogNegative) AND iConvCtrl.Cmd.PrintMark ) THEN
				iVa_RecPrintPosition := gAx_Master.Out.Position;
			END_IF

			IF (iVa_RecPrintPosition - gAx_Master.Out.Position) > (PRINT_MARK_LIMIT) AND iVa_RecPrintPosition <> K_ZERO THEN
				gAx_Master.In.JogNegative := FALSE;
				iConvCtrl.Cmd.JogBack := FALSE;
				MasterStep := MANUAL;
			ELSE
				iConvCtrl.Status.JogNegReady := TRUE;
			END_IF

	END_CASE

	iConvCtrl.Cmd.PrintMark := gAx_Slave.Out.Info.DigitalInputsStatus.Trigger1;
	iVa_SetMasterInputs.Axis := ADR(gAxis01);
	iVa_SetMasterInputs.Enable := TRUE;
	iVa_SetMasterInputs.HomeSwitch := gAx_Slave.Out.Info.DigitalInputsStatus.Trigger1;
	iVa_SetMasterInputs();

END_PROGRAM

PROGRAM _EXIT
	(* Insert code here *)

END_PROGRAM
```

### Package Logical/InfraStructure - Infrastructure Package

### Package Logical/InfraStructure/Alarm - Alarm Package

### Program Logical/InfraStructure/Alarm/Alarm (IEC) - Alarm Task

#### Variables.var
```iecst
VAR
	iFB_Alarm : MpAlarmXCore; (*MpAlarmXcore FB*)
END_VAR
```

#### Main.st
```iecst
(*********************************************************************************
 * Copyright: B&R Industrial Automation GmbH
 * Author:    kasliwals
 * Created:   December 16, 2023/11:54 PM
* Description: Alarm Configuration
* Version : 1.0.0.0
 *********************************************************************************)

PROGRAM _INIT
	(* Insert code here *)

END_PROGRAM

PROGRAM _CYCLIC
	(* Insert code here *)
	iFB_Alarm.Enable := TRUE;
	iFB_Alarm.MpLink := ADR(gAlarmXMain);

	iFB_Alarm();

END_PROGRAM

PROGRAM _EXIT
	(* Insert code here *)
	iFB_Alarm.Enable := FALSE;
	iFB_Alarm();

END_PROGRAM
```

- Visualisation Logical/InfraStructure/Visu (not shown)

- Visualisation Logical/mappView (not shown)

Listed in the project but not available here: Logical/Global.typ, Logical/Axis/acp10etxen, Logical/InfraStructure/Documentation
